FUNCTION_BLOCK SENSOR_COUNTER
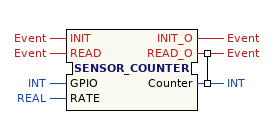
  EVENT_INPUT
    INIT;
    READ;
  END_EVENT
  EVENT_OUTPUT
    INIT_O;
    READ_O WITH Counter;
  END_EVENT
  VAR_INPUT
    GPIO : INT;
    RATE : REAL;
  END_VAR
  VAR_OUTPUT
    Counter : INT;
  END_VAR
END_FUNCTION_BLOCK
